{attribute addProperty BoxType "EK1122-0000-0018"}
{attribute addProperty Id "Beckhoff_EL25xxsub_EK1100EK1100_179A0949162"}
{attribute addProperty CRC "1736503315"}
{attribute addProperty SizeInBites "16"}
{attribute addProperty SizeInBytes "2"}
TYPE Beckhoff_EL25xxEK1122_6780F013 EXTENDS EK1122_179A0949 :
STRUCT
	{attribute addProperty Name "Beckhoff_EL25xxsub_EK1100"}
	Beckhoff_EL25xxsub_EK1100 : EK1100_179A0949;
END_STRUCT
END_TYPE

(* stored: Version 1.2.0.0, ProductVersion 3.1.4024.9
   DUT Beckhoff_EL25xxEK1122_6780F013: Id {6330d8e3-146a-4f42-9e6f-08140386259d} *)
